// TIA Portal V18 export
DATA_BLOCK "SS1_CPU1214_AI_Vars"   // DB11011
{ S7_Optimized_Access := 'FALSE' }
VERSION : 0.1
// stored: AutoNumber false, DBAccessibleFromOPCUA true, IsOnlyStoredInLoadMemory false, IsWriteProtectedInAS false
   VAR
      AI1 { S7_SetPoint := 'True'} : "UDT_AIadv";   // AHU NF Перепад тиску повітря (2.40)
      AI2 { S7_SetPoint := 'True'} : "UDT_AIadv";   // HS Вихід нагрівача (10.11)
   END_VAR
BEGIN
   AI1.rValue := 368.9236;
   AI1.rMin := 0.0;
   AI1.rMax := 50000.0;
   AI1.rCalibration := 0.0;
   AI1.iFuncSystemID := 2;
   AI1.iFuncVar := 2;
   AI1.rFilterSet := 0.0;
   AI2.rValue := 0.0;
   AI2.rMin := 0.0;
   AI2.rMax := 0.0;
   AI2.rCalibration := 0.0;
   AI2.iFuncSystemID := 10;
   AI2.iFuncVar := 7;
   AI2.rFilterSet := 0.0;
END_DATA_BLOCK
